(* IEC 61131-3 sources: automatic-screwdriver-line/src/POU/Actuators, 4 files *)

(* ---- FB_Cobot.st ---- *)
// Generated from Automatic_ScrewDriver_Line.xml by tools/export_st.py - do not edit.
// The CODESYS project is the source of truth.

FUNCTION_BLOCK FB_Cobot EXTENDS FB_FunctionBlock_Base IMPLEMENTS I_Mover
VAR_INPUT
	MoverPosEcho : INT;   // Echo to ensure synchronisation with MoverTarget
	MoverDone : BOOL;
	MoverHeartbeat : INT;   // Watchdog counter to make sure Cobot connection is not lost
END_VAR
VAR_OUTPUT
	MoverEnable : BOOL;
	MoverTarget : INT;
	MoverExecute : BOOL;
END_VAR
VAR
	_state : MoverState := MoverState.Idle;
	_TimerEcho : TON;
	_TimerMove : TON;
	_TimerEnablement : TON;
	_LastHeartbeat : INT;
	_HbTimer : TON;
	_Alive : BOOL;
	_HbChanged : BOOL;
END_VAR

METHOD Reset : BOOL

ClearError();
Disable();
MoverTarget :=  0;
_state := MoverState.Idle;
_TimerEnablement(IN := FALSE, PT := T#1S);
_TimerEcho(IN := FALSE, PT := T#2S);
_TimerMove(IN := FALSE, PT := T#30S);
_HbTimer(IN := FALSE, PT := T#500MS);

Reset := TRUE;
END_METHOD

METHOD MoveToPosition : BOOL
VAR_INPUT
	Position : REAL;
END_VAR

MoveToPosition := FALSE;

CASE _state OF

	MoverState.Idle:
		// Never start a cycle while the robot still asserts Done from a previous one
		IF NOT MoverDone THEN
			MoverTarget  := REAL_TO_INT(Position * 10.0);
			MoverExecute := FALSE;
			_state := MoverState.WaitingEcho;
		END_IF

	MoverState.WaitingEcho:
		IF MoverPosEcho = MoverTarget THEN
			MoverExecute := TRUE;
			_state := MoverState.Moving;
		ELSIF _TimerEcho.Q THEN
			RaiseError(ErrorCode.CobotNotConnected);
		END_IF

	MoverState.Moving:
		IF MoverDone THEN
			MoverExecute := FALSE;
			_state := MoverState.WaitingDoneReleased;
		ELSIF _TimerMove.Q THEN
			RaiseError(ErrorCode.CobotMovementNotReached);
		END_IF

	MoverState.WaitingDoneReleased:
		IF NOT MoverDone THEN
			MoveToPosition := TRUE;
			_state := MoverState.Idle;
		END_IF

END_CASE

_TimerEcho(IN := (_state = MoverState.WaitingEcho), PT := T#2S);
_TimerMove(IN := (_state = MoverState.Moving), PT := T#30S);
END_METHOD

METHOD Enable : BOOL

_HbChanged := (MoverHeartbeat <> _LastHeartbeat);
_LastHeartbeat := MoverHeartbeat;
_HbTimer(IN := NOT _HbChanged, PT := T#500MS);
_Alive := NOT _HbTimer.Q;

Enable := FALSE;
MoverEnable := TRUE;

_TimerEnablement(IN := NOT _Alive, PT := T#1S);

IF _Alive THEN
	Enable := TRUE;
ELSIF _TimerEnablement.Q THEN
	RaiseError(ErrorCode.CobotNotConnected);
END_IF
END_METHOD

METHOD Disable : BOOL

MoverEnable  := FALSE;
MoverExecute := FALSE;
Disable := TRUE;
END_METHOD

END_FUNCTION_BLOCK

(* ---- FB_ConveyorElectrical.st ---- *)
// Generated from Automatic_ScrewDriver_Line.xml by tools/export_st.py - do not edit.
// The CODESYS project is the source of truth.

FUNCTION_BLOCK FB_ConveyorElectrical EXTENDS FB_FunctionBlock_Base IMPLEMENTS I_Mover
VAR_INPUT
	MoverActPos : REAL;
	MoverReady : BOOL;
END_VAR
VAR_OUTPUT
	MoverEnable : BOOL;
	MoverExecuteFor : BOOL;
	MoverExecuteBac : BOOL;
END_VAR
VAR
	_MoverTarget : REAL;
	_TimerEnablement : TON;
	_TimerMoveLinear : TON;
END_VAR

METHOD Reset : BOOL

ClearError();
Disable();
MoverExecuteFor := FALSE;
MoverExecuteBac := FALSE;
_MoverTarget :=  0.0;
_TimerEnablement(IN := FALSE, PT := T#1S);
_TimerMoveLinear(IN := FALSE, PT := T#100S);
Reset := TRUE;
END_METHOD

METHOD MoveToPosition : BOOL
VAR_INPUT
	Position : REAL;
END_VAR

MoveToPosition := FALSE;

_MoverTarget := Position;

IF _TimerMoveLinear.Q THEN
	RaiseError(ErrorCode.TargetNotReached);
ELSIF _MoverTarget - MoverActPos >= 1 THEN
	MoverExecuteFor := TRUE;
ELSIF _MoverTarget - MoverActPos <= -1 THEN
	MoverExecuteBac := TRUE;
ELSE
	MoveToPosition := TRUE;
	MoverExecuteFor := FALSE;
	MoverExecuteBac := FALSE;
END_IF

_TimerMoveLinear(IN := (MoverExecuteFor OR MoverExecuteBac), PT := T#100S);
END_METHOD

METHOD Enable : BOOL

Enable := FALSE;

MoverEnable := TRUE;
_TimerEnablement(IN := MoverEnable AND NOT MoverReady, PT := T#1S);

IF MoverReady THEN
	Enable := TRUE;
ELSIF _TimerEnablement.Q THEN
	RaiseError(ErrorCode.EnablementError);
END_IF
END_METHOD

METHOD Disable : BOOL

MoverEnable := FALSE;
Disable := TRUE;
END_METHOD

END_FUNCTION_BLOCK

(* ---- FB_Spindle.st ---- *)
// Generated from Automatic_ScrewDriver_Line.xml by tools/export_st.py - do not edit.
// The CODESYS project is the source of truth.

FUNCTION_BLOCK FB_Spindle EXTENDS FB_FunctionBlock_Base IMPLEMENTS I_Actuator
VAR_INPUT
	SpeedDegPerSec : DINT := Machine_Constants.TOOL_SPEED;
	SpindleReady : BOOL;
	SpindleDone : BOOL;
END_VAR
VAR_OUTPUT
	SpindleEnable : BOOL;
	SpindleExecute : BOOL;
	SpindleExecuteTime : TIME;
END_VAR
VAR
	_AngleTarget : DINT;
	_Started : BOOL;
	_TimerEnablement : TON;
	_TimerProcessTool : TON;
END_VAR

METHOD Reset : BOOL

ClearError();
Disable();
SpindleEnable := FALSE;
SpindleExecute := FALSE;
SpindleExecuteTime := T#0S;
_AngleTarget := 0;
_Started := FALSE;
_TimerEnablement(IN := FALSE, PT := T#1S);
_TimerProcessTool(IN := FALSE, PT := T#20S);
Reset := TRUE;
END_METHOD

METHOD ProcessTool : BOOL
VAR_INPUT
	Angle : DINT;
END_VAR

ProcessTool := FALSE;
_TimerProcessTool(IN := SpindleExecute AND NOT SpindleDone, PT := T#20S);
_AngleTarget := ABS(Angle);

IF NOT _Started AND SpindleEnable THEN
	SpindleExecuteTime := DINT_TO_TIME(_AngleTarget*1000/SpeedDegPerSec);
	SpindleExecute := TRUE;
	_Started := TRUE;
ELSIF SpindleDone THEN
	SpindleExecute := FALSE;
	_Started := FALSE;
	ProcessTool := TRUE;
ELSIF _TimerProcessTool.Q THEN
	RaiseError(ErrorCode.SpindleError);
END_IF
END_METHOD

METHOD Enable : BOOL

Enable := FALSE;

SpindleEnable := TRUE;
_TimerEnablement(IN := SpindleEnable AND NOT SpindleReady, PT := T#1S);

IF SpindleReady THEN
	Enable := TRUE;
ELSIF _TimerEnablement.Q THEN
	RaiseError(ErrorCode.EnablementError);
END_IF
END_METHOD

METHOD Disable : BOOL

SpindleEnable := FALSE;
Disable := TRUE;
END_METHOD

END_FUNCTION_BLOCK

(* ---- FB_zAxis.st ---- *)
// Generated from Automatic_ScrewDriver_Line.xml by tools/export_st.py - do not edit.
// The CODESYS project is the source of truth.

FUNCTION_BLOCK FB_zAxis EXTENDS FB_FunctionBlock_Base
VAR_INPUT
	zDown : BOOL;
	ScrewEngaged : BOOL;
	ScrewReleased : BOOL;
END_VAR
VAR_OUTPUT
	zValve : BOOL;
END_VAR
VAR
	_timerUp : TON;
	_timerDown : TON;
END_VAR

METHOD Reset : BOOL

ClearError();

zValve := FALSE;

IF zDown THEN
	Reset := TRUE;
END_IF

_timerUp(IN := FALSE, PT := T#5S);
_timerDown(IN := FALSE, PT := T#5S);
END_METHOD

METHOD Engage : ActionResult

Engage := ActionResult.Busy;
zValve := TRUE;

_timerUp(IN := zValve AND NOT ScrewEngaged, PT := T#5S);
_timerDown(IN := FALSE, PT := T#5S);

IF ScrewEngaged THEN
	Engage := ActionResult.Done;
ELSIF _timerUp.Q THEN
	Engage := ActionResult.Failed;
END_IF
END_METHOD

METHOD Retract : BOOL

Retract := FALSE;
zValve := FALSE;

_timerDown(IN := NOT zValve AND NOT (zDown AND ScrewReleased), PT := T#5S);
_timerUp(IN := FALSE, PT := T#5S);

IF zDown AND ScrewReleased THEN
    Retract := TRUE;
ELSIF _timerDown.Q THEN
	RaiseError(ErrorCode.ScrewNotReleased);
END_IF
END_METHOD

END_FUNCTION_BLOCK
